FUNCTION_BLOCK FB_BARRIDOXY
VAR_INPUT
	speed : REAL;
END_VAR
VAR_OUTPUT
	Xbarrido: REAL := 0;
	Ybarrido : REAL :=1000;
END_VAR
VAR
END_VAR

IF Xbarrido < 500 THEN
	Xbarrido:=Xbarrido+speed;
	ELSE
		Xbarrido := -500;
		Ybarrido:=Ybarrido+speed;
	END_IF
	
IF Ybarrido > 2000 THEN
	Ybarrido := 1000;
END_IF

END_FUNCTION_BLOCK

(* stored: Version 1.1.0.1, ProductVersion 3.1.4024.4
   POU FB_BARRIDOXY: Id {d35cf1a9-8eea-43ee-87cc-45ae10fa1aa6}, SpecialFunc None *)
